{attribute 'GeneratedUsingTerminal: EKM1101-0000-0016'}
{attribute addProperty BoxType "EKM1101-0000-0016"}
{attribute addProperty Id "StatusAT %I*Status_F2CE6D917ValueAT %I*REAL4"}
{attribute addProperty CRC "1624595570"}
{attribute addProperty Size "11"}
TYPE MMS_Voltage_Up_Out_Inputs_60D55C72 EXTENDS InputBase_8311D824 :
STRUCT
	{attribute addProperty Name "Status"}
	Status AT %I* : Status_F2CE6D91;
	{attribute addProperty Name "Value"}
	Value AT %I* : REAL;
END_STRUCT
END_TYPE

(* stored: Version 1.2.0.0, ProductVersion 3.1.4024.11
   DUT MMS_Voltage_Up_Out_Inputs_60D55C72: Id {7dac000e-e7d7-46d4-8f07-5ea3df92f456} *)
